# EPICS substitutions: examples/test/el6080/ecmcEL6080_app_ints.substitutions
file "ecmcEL6080_app_ints.template"
{
  pattern {EC_TYPE}
          {U8     }
          {S8     }
          {U16     }
          {S16     }
          {U32     }
          {S32     }
}
